FUNCTION LogToWarning : BOOL
VAR_INPUT
	msgFmtStr : T_MaxString;
	messageArg : T_MaxString;
END_VAR
VAR
END_VAR

ADSLOGSTR(msgCtrlMask := ADSLOG_MSGTYPE_WARN, msgFmtStr := msgFmtStr, strArg := messageArg);

END_FUNCTION

(* stored: Version 1.1.0.1, ProductVersion 3.1.4024.12
   POU LogToWarning: Id {571806e4-e2af-42f9-a605-12d063811f93}, SpecialFunc None *)
